{attribute 'Tc2GvlVarNames'}
VAR_GLOBAL

	Start_mesure_Barre:BOOL:=FALSE;

	Time_Recul_Mesure_Barre:TIME:=t#5s;
	Mesure_Barre_Ok:BOOL:=FALSE;
	Fin_Desserage_Pince:BOOL:=FALSE;
	Fin_Serrage_Pince:BOOL:=FALSE;
	X_Cell_Mesure_Barre:LREAL;

	Time_Serr_Dess_Pince:TIME;

	B_Voyant_Pince:BOOL:=FALSE;
	Pos_X_Mesure_Barre:LREAL;
	
	Bit_Relevage_pince: BOOL;
	Bit_Abaissement_pince: BOOL;
	Dem_Relevage_auto	:BOOL;
	
	Cde_Serrage_Desserrage	:BOOL;
	Dem_Serrage,Dem_Desserrage	:BOOL;

	Zone_X_Interdit_decoupe		:REAL; //Correspond à la distance entre le fd de pince et l'extremité de celle ci une fois ouverte, à mesurer
	Pince_interdit_decoupe		:BOOL;	// Défaut si le laser est trop proche du chariot en manu

END_VAR

(* stored: Version 1.1.0.1
   GVL Global_Chariot: Id {ad69e8d5-d28c-4935-a0bf-bfec9a41b1eb} *)
